% RSLogix 500 project P5_KOBIERSKI_M.RSS, saved by version 8.30.00.16 %
PROJECT "UNTITLED"    % processor: Bul.1763 MicroLogix 1100 Series B %

PROGRAM FILES
  LAD 2 "MAIN"  4 rungs
  LAD 3 "INPUT"  3 rungs
  LAD 4 "CTRL"  5 rungs

DATA FILES
  O0 OUTPUT  4 elements
  I1 INPUT  6 elements
  S2 STATUS  66 elements
  B3 BINARY  1 elements
  T4 TIMER  2 elements
  C5 COUNTER  1 elements
  R6 CONTROL  1 elements
  N7 INTEGER  1 elements
  F8 FLOAT  3 elements

LADDER 2 "MAIN"
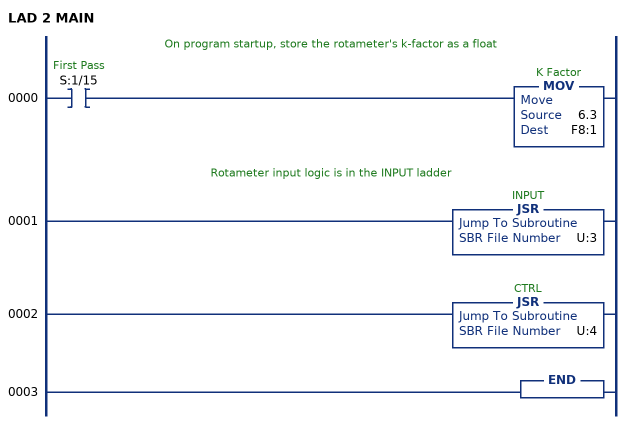
% Rung: 0 %
% On program startup, store the rotameter's k-factor as a float %
SOR XIC S:1/15 MOV 6.3 F8:1 EOR
%   S:1/15  "First Pass" %
%   F8:1  "K Factor" %
% Rung: 1 %
% Rotameter input logic is in the INPUT ladder %
SOR JSR U:3 EOR
%   U:3  "INPUT" %
% Rung: 2 %
SOR JSR U:4 EOR
%   U:4  "CTRL" %
% Rung: 3 %
SOR END EOR

LADDER 3 "INPUT"
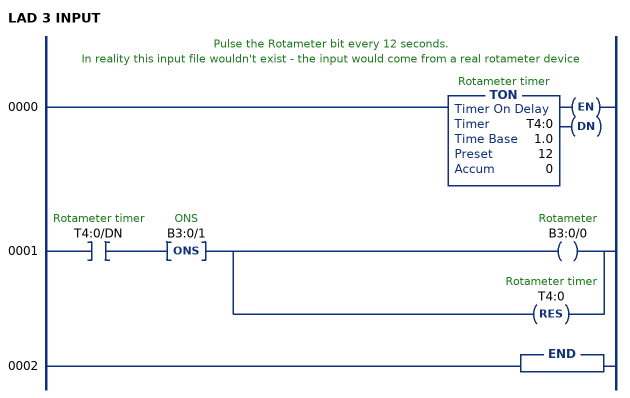
% Rung: 0 %
% Pulse the Rotameter bit every 12 seconds.
% In reality this input file wouldn't exist - the input would come from a real rotameter device %
SOR TON T4:0 1.0 12 0 EOR
%   T4:0  "Rotameter timer" %
% Rung: 1 %
SOR XIC T4:0/DN ONS B3:0/1 BST OTE B3:0/0 NXB RES T4:0 BND EOR
%   T4:0  "Rotameter timer" %
%   B3:0/1  "ONS" %
%   B3:0/0  "Rotameter" %
% Rung: 2 %
SOR END EOR

LADDER 4 "CTRL"
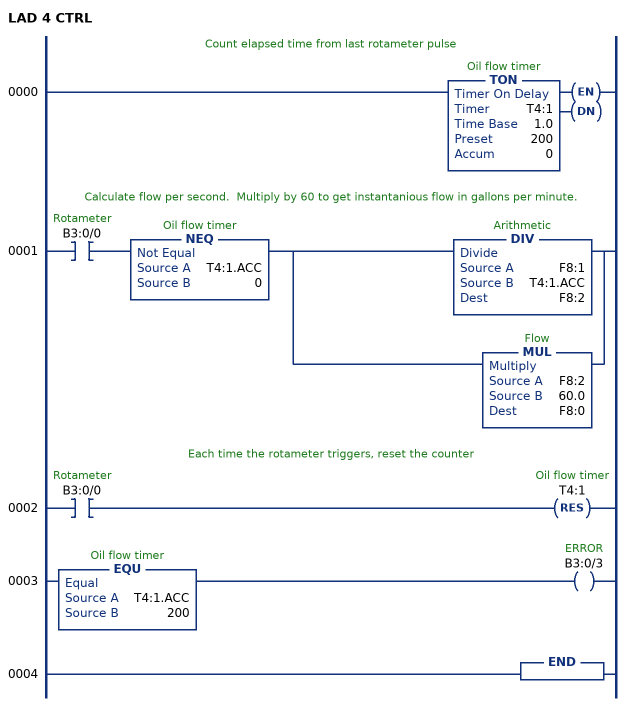
% Rung: 0 %
% Count elapsed time from last rotameter pulse %
SOR TON T4:1 1.0 200 0 EOR
%   T4:1  "Oil flow timer" %
% Rung: 1 %
% Calculate flow per second.  Multiply by 60 to get instantanious flow in gallons per minute. %
SOR XIC B3:0/0 NEQ T4:1.ACC 0 BST DIV F8:1 T4:1.ACC F8:2 NXB MUL F8:2 60.0 F8:0 BND EOR
%   B3:0/0  "Rotameter" %
%   T4:1  "Oil flow timer" %
%   F8:1  "K Factor" %
%   F8:2  "Arithmetic" %
%   F8:0  "Flow" %
% Rung: 2 %
% Each time the rotameter triggers, reset the counter %
SOR XIC B3:0/0 RES T4:1 EOR
%   B3:0/0  "Rotameter" %
%   T4:1  "Oil flow timer" %
% Rung: 3 %
SOR EQU T4:1.ACC 200 OTE B3:0/3 EOR
%   T4:1  "Oil flow timer" %
%   B3:0/3  "ERROR" %
% Rung: 4 %
SOR END EOR

OTHER DOCUMENTED ADDRESSES
  B3:0/2  "Running"
  C5:0  "Oil flow time"
  U:5  "PULSE"

DATA TABLE (non-zero values as saved)
DATA T4
% .PRE .ACC %
% T4:0 % 12 0
% T4:1 % 200 0
DATA C5
% .PRE .ACC %
% C5:0 % 200 0
